TYPE ST_Welding_Control_Circle_86s_Input :
STRUCT
	t: LREAL;
END_STRUCT
END_TYPE

(* stored: Version 1.1.0.1, ProductVersion 3.1.4020.12
   DUT ST_Welding_Control_Circle_86s_Input: Id {55767307-b0a6-4769-9cac-24249d060546} *)
